// TIA Portal V19 export
FUNCTION_BLOCK "GBL_TandD"   // FB20, LAD
{ S7_Optimized_Access := 'TRUE' }
// stored: MemoryReserve 100, SetENOAutomatically false
   VAR
      "write time" { ExternalAccessible := 'False'; ExternalVisible := 'False'; ExternalWritable := 'False'} : DTL;
      "System Time" { ExternalAccessible := 'False'; ExternalVisible := 'False'; ExternalWritable := 'False'} : DTL;
   END_VAR
   VAR_TEMP   // added for the SCL form of the ladder/FBD networks
      _w1 : Bool;
   END_VAR
BEGIN

REGION Network 1
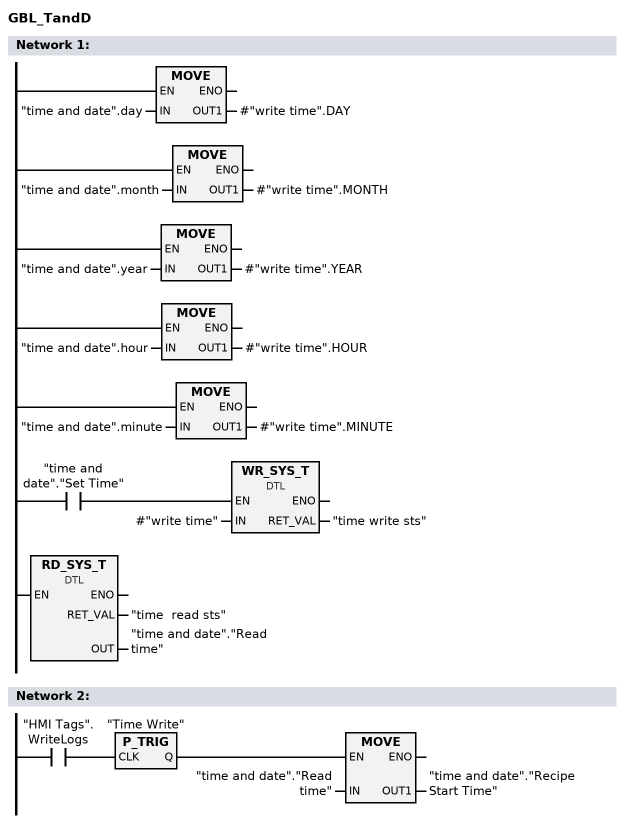
   RUNG wire#powerrail
      Move(in := "time and date".day, out1 => #"write time".DAY)
   END_RUNG
   RUNG wire#powerrail
      Move(in := "time and date".month, out1 => #"write time".MONTH)
   END_RUNG
   RUNG wire#powerrail
      Move(in := "time and date".year, out1 => #"write time".YEAR)
   END_RUNG
   RUNG wire#powerrail
      Move(in := "time and date".hour, out1 => #"write time".HOUR)
   END_RUNG
   RUNG wire#powerrail
      Move(in := "time and date".minute, out1 => #"write time".MINUTE)
   END_RUNG
   RUNG wire#powerrail
      Contact( "time and date"."Set Time" )
      { S7_Templates := "date_type := DTL" } WR_SYS_T(IN := #"write time", RET_VAL => "time write sts")
   END_RUNG
   RUNG wire#powerrail
      { S7_Templates := "date_type := DTL" } RD_SYS_T(RET_VAL => "time  read sts", OUT => "time and date"."Read time")
   END_RUNG
   // the same network as SCL:
   #"write time".DAY := "time and date".day;
   #"write time".MONTH := "time and date".month;
   #"write time".YEAR := "time and date".year;
   #"write time".HOUR := "time and date".hour;
   #"write time".MINUTE := "time and date".minute;
   IF "time and date"."Set Time" THEN "time write sts" := WR_SYS_T(IN := #"write time"); END_IF;
   "time  read sts" := RD_SYS_T(OUT => "time and date"."Read time");
END_REGION

REGION Network 2
   RUNG wire#powerrail
      Contact( "HMI Tags".WriteLogs )
      P_Trig( "Time Write" )
      Move(in := "time and date"."Read time", out1 => "time and date"."Recipe Start Time")
   END_RUNG
   // the same network as SCL:
   #_w1 := "HMI Tags".WriteLogs AND NOT "Time Write";   // rising edge
   "Time Write" := "HMI Tags".WriteLogs;
   IF #_w1 THEN "time and date"."Recipe Start Time" := "time and date"."Read time"; END_IF;
END_REGION
END_FUNCTION_BLOCK
